// TIA Portal V16 export
// export: Created 2024-03-28T09:48:20.9146827Z, ExportSetting WithDefaults, DisplayName Totally Integrated Automation Portal, DisplayVersion V16, DisplayName TIA Portal Version Control Interface, DisplayVersion V16, DisplayName TIA Portal Openness, DisplayVersion V16, DisplayName STEP 7 Professional, DisplayVersion V16, DisplayName STEP 7 Safety, DisplayVersion V16, DisplayName WinCC Advanced, DisplayVersion V16
TYPE "UR_9_O2T_Registers"
// stored: IsFailsafeCompliant false
   STRUCT
      Bits { S7_SetPoint := 'True'} : "UR__O2T_bits";
      Ints { S7_SetPoint := 'True'} : "UR__O2T_ints";
      Floats { S7_SetPoint := 'True'} : "UR__O2T_floats";
   END_STRUCT;
END_TYPE
